// TwinCAT 3 PLC project ManRiding
// ProgramVersion: 3.1.4023.0
// libraries:
//   Tc2_ControllerToolbox, * (Beckhoff Automation GmbH)
//   Tc2_Math, * (Beckhoff Automation GmbH)
//   Tc2_MC2, * (Beckhoff Automation GmbH)
//   Tc2_MC2_Drive, * (Beckhoff Automation GmbH)
//   Tc2_ModbusSrv, * (Beckhoff Automation GmbH)
//   Tc2_SerialCom, * (Beckhoff Automation GmbH)
//   Tc2_Standard, * (Beckhoff Automation GmbH)
//   Tc2_System, * (Beckhoff Automation GmbH)
//   Tc2_TcpIp, * (Beckhoff Automation GmbH)
//   Tc2_Utilities, * (Beckhoff Automation GmbH)
//   Tc3_Database, * (Beckhoff Automation GmbH)
//   Tc3_JsonXml, * (Beckhoff Automation GmbH)
//   Tc3_Module, * (Beckhoff Automation GmbH)
//   VisuDialogs, * (System)
//   VisuSymbols, * (System)
//   VisuSymbols,3.5.10.0,System
// project tree:
//   / GlobalTextList.TcGTLO, PlcTask.TcTTO, Visualization Manager.TcVMO (not stored)
//   GVLs/ GVL.TcGVL, INPUT.TcGVL, OUTPUT.TcGVL
//   POUs/ FB_AxisControl.TcPOU, FUN_In_Zone.TcPOU, MAIN.TcPOU
//   VISUs/ Visualization.TcVIS
// real-time tasks:
//   TASK PlcTask: cycle T#10ms, priority 20, ADS port 350
// motion (NC):
//   TASK NC-Task 1 SAF: cycle T#2ms, priority 4, ADS port 501
//   TASK NC-Task 1 SVB: cycle T#10ms, priority 8, ADS port 511
//   AXIS Axis 1 (BogieDrv1) (id 1)
//     OtherSettings: AllowMotionCmdToSlave=true
//     encoder EncType=1
//     drive DrvType=5
//       Analog: TorqueSetpointScale=10, ScaleFactorActTorque=0.1
//     controller CtrType=1
//       CtrPara: PriorControlFactor=1
//         Observer: BandWidth=20
//   AXIS Axis 2 (BogieDrv2) (id 2)
//     OtherSettings: AllowMotionCmdToSlave=true
//     encoder EncType=1
//     drive DrvType=5
//       Analog: TorqueSetpointScale=10, ScaleFactorActTorque=0.1
//     controller CtrType=1
//       CtrPara: PriorControlFactor=1
//         Observer: BandWidth=20
//   AXIS Axis 3 (BogieDrv3) (id 3)
//     OtherSettings: AllowMotionCmdToSlave=true
//     encoder EncType=1
//     drive DrvType=5
//       Analog: TorqueSetpointScale=10, ScaleFactorActTorque=0.1
//     controller CtrType=1
//       CtrPara: PriorControlFactor=1
//         Observer: BandWidth=20
//   AXIS Axis 4 (BogieDrv4) (id 4)
//     OtherSettings: AllowMotionCmdToSlave=true
//     encoder EncType=1
//     drive DrvType=5
//       Analog: TorqueSetpointScale=10, ScaleFactorActTorque=0.1
//     controller CtrType=1
//       CtrPara: PriorControlFactor=1
//         Observer: BandWidth=20
//   AXIS Axis 5 (Stabiliser A) (id 5)
//     Dynamic: AccelerationMaximum=50000, DecelerationMaximum=50000, Acceleration=1371.32, Deceleration=1371.32, Jerk=1385020, FastAxisStopSignalType=4
//     Velo: RefSearch=1.357738094695, RefSync=1.357738094695, SlowManual=6.788690473475, FastManual=40.73214284085, Fast=135.7738094695, Maximum=135.774
//     OtherSettings: AllowMotionCmdToSlave=true
//     encoder EncType=19
//       EncPara: ScaleFactorNumerator=3.57142857, ScaleFactorDenominator=1048576, Offset=104.9, MaxCount=#xffffffff
//         SoftEndMinControl: Enable=true, Range=-10
//         SoftEndMaxControl: Enable=true, Range=200
//     drive DrvType=16
//       DrvPara: MaxCount=#xffffffff, DriveControlDWord=#x00020000
//         Analog: VeloReferenz=149.35119041645, VeloScale=32, TorqueSetpointScale=10, ScaleFactorActTorque=0.1
//         TimeComp: TaskDelayCycles=1
//     controller CtrType=1
//       CtrPara: PriorControlFactor=1
//         PosDiffControl: Enable=false
//         PID: PosKp=30
//         Observer: BandWidth=20
//   AXIS Axis 6 (Stabiliser B) (id 6)
//     Dynamic: AccelerationMaximum=50000, DecelerationMaximum=50000, Acceleration=1371.32, Deceleration=1371.32, Jerk=1385030, FastAxisStopSignalType=4
//     Velo: RefSearch=1.357738094695, RefSync=1.357738094695, SlowManual=6.788690473475, FastManual=40.73214284085, Fast=135.7738094695, Maximum=135.774
//     OtherSettings: AllowMotionCmdToSlave=true
//     encoder EncType=19
//       EncPara: ScaleFactorNumerator=3.57142857, ScaleFactorDenominator=1048576, Offset=411, Inverse=true, MaxCount=#xffffffff
//         SoftEndMinControl: Enable=true, Range=-10
//         SoftEndMaxControl: Enable=true, Range=200
//     drive DrvType=16
//       DrvPara: Inverse=true, MaxCount=#xffffffff, DriveControlDWord=#x00020000
//         Analog: VeloReferenz=149.35119041645, VeloScale=32, TorqueSetpointScale=10, ScaleFactorActTorque=0.1
//         TimeComp: TaskDelayCycles=1
//     controller CtrType=1
//       CtrPara: PriorControlFactor=1
//         PosDiffControl: Enable=false
//         PID: PosKp=30
//         Observer: BandWidth=20
//   AXIS Axis 7 (Stabiliser C) (id 7)
//     Dynamic: AccelerationMaximum=50000, DecelerationMaximum=50000, Acceleration=1371.32, Deceleration=1371.32, Jerk=1385030, FastAxisStopSignalType=4
//     Velo: RefSearch=1.357738094695, RefSync=1.357738094695, SlowManual=6.788690473475, FastManual=40.73214284085, Fast=135.7738094695, Maximum=135.774
//     OtherSettings: AllowMotionCmdToSlave=true
//     encoder EncType=19
//       EncPara: ScaleFactorNumerator=3.57142857, ScaleFactorDenominator=1048576, Offset=-4435, MaxCount=#xffffffff
//         SoftEndMinControl: Enable=true, Range=-10
//         SoftEndMaxControl: Enable=true, Range=200
//     drive DrvType=16
//       DrvPara: MaxCount=#xffffffff, DriveControlDWord=#x00020000
//         Analog: VeloReferenz=149.35119041645, VeloScale=32, TorqueSetpointScale=10, ScaleFactorActTorque=0.1
//         TimeComp: TaskDelayCycles=1
//     controller CtrType=1
//       CtrPara: PriorControlFactor=1
//         PosDiffControl: Enable=false
//         PID: PosKp=30
//         Observer: BandWidth=20
//   AXIS Axis 8 (Stabiliser D) (id 8)
//     Dynamic: AccelerationMaximum=50000, DecelerationMaximum=50000, Acceleration=1371.32, Deceleration=1371.32, Jerk=1385030, FastAxisStopSignalType=4
//     Velo: RefSearch=1.357738094695, RefSync=1.357738094695, SlowManual=6.788690473475, FastManual=40.73214284085, Fast=135.7738094695, Maximum=135.774
//     OtherSettings: AllowMotionCmdToSlave=true
//     encoder EncType=19
//       EncPara: ScaleFactorNumerator=3.57142857, ScaleFactorDenominator=1048576, Offset=288.9, Inverse=true, MaxCount=#xffffffff
//         SoftEndMinControl: Enable=true, Range=-10
//         SoftEndMaxControl: Enable=true, Range=200
//     drive DrvType=16
//       DrvPara: Inverse=true, MaxCount=#xffffffff
//         Analog: VeloReferenz=149.35119041645, VeloScale=32, TorqueSetpointScale=10, ScaleFactorActTorque=0.1
//         TimeComp: TaskDelayCycles=1
//     controller CtrType=1
//       CtrPara: PriorControlFactor=1
//         PosDiffControl: Enable=false
//         PID: PosKp=30
//         Observer: BandWidth=20

CONFIGURATION ManRiding
    RESOURCE PLC ON TwinCAT3
        TASK PlcTask(INTERVAL := T#10ms, PRIORITY := 20);
        PROGRAM MAIN WITH PlcTask : MAIN;
    END_RESOURCE
END_CONFIGURATION

// ---- GVLs/GVL.TcGVL
	{attribute 'qualified_only'}
	{attribute 'TcContextName':='PlcTaskMAIN'}
VAR_GLOBAL PERSISTENT
	//New Version
	Bogie_Clean_Position : REAL := 0;
		
END_VAR

VAR_GLOBAL CONSTANT
	
END_VAR


VAR_GLOBAL
	Home_Button_Activated 		: BOOL := FALSE;
	Cleaning_Button_Activated 	: BOOL := FALSE;
	Finish_Current_Brick 		: BOOL := FALSE;
	HMI_Connected 				: BOOL := FALSE;
	database		: ARRAY[0..100] OF STRING(100);(* Target PLC database *)

	
	AMSID : T_AmsNetId  := '5.61.32.144.1.1';       // this is the ADS address for the IPC on the robot

	Use_Current_As_Clean_Position : BOOL := FALSE;
	
{region "axis refs"}	
	Bogie_DriveA	: AXIS_REF; 
	Bogie_DriveB	: AXIS_REF; 
	Bogie_DriveC	: AXIS_REF; 
	Bogie_DriveD	: AXIS_REF; 		 
	Stabiliser_A_Axis	: AXIS_REF;
	Stabiliser_B_Axis	: AXIS_REF;	
	Stabiliser_C_Axis	: AXIS_REF;		
	Stabiliser_D_Axis	: AXIS_REF;		
		 
	Bogie_DriveA_Velocity        	: LREAL;
	Bogie_DriveB_Velocity        	: LREAL;
	Bogie_DriveC_Velocity        	: LREAL;
	Bogie_DriveD_Velocity        	: LREAL;

{endregion}
	 
{region "TCP/Lazer Adjust"}

{endregion}

{region "Bogie Alarm"}
	BogieAlarmTimer : TON := (PT := T#2S);
{endregion}
	
{region "procedure variables"}	
	// Main procedure Variables
	IsEnabled		   : BOOL	:= FALSE;
	Is_Running          : BOOL;                         // the boolean to indicate if the robot is running in a sequence mode
	Is_Start_Button_Pressed          : BOOL;                         // boolean representing the start button on the HMI
	Is_Stop_Button_Pressed           : BOOL := TRUE;                 // boolean representing the stop button on the HMI - boots to false, preventing the sequence initiaiting without explicit commmand
	Cancel_Manuals					 : BOOL;		 
	
{region "ablr/ bogie vars"}	
	// Four Wheel Drive Bogie System
	Bogie_Pause					: BOOL := FALSE;
	  
	Bogie_DriveA_Current_Position      : REAL;                          // bogie current position  
	Bogie_DriveA_Required_Position     : REAL;
	Bogie_DriveA_In_Position           : BOOL;
	Bogie_DriveA_Manual_Enable         : BOOL;
	Bogie_DriveA_Encoder_Reset         : BOOL := FALSE;
	Bogie_DriveA_Pause					: BOOL := FALSE;
		 
	Bogie_DriveB_Current_Position      : REAL;                          // bogie current position
	Bogie_DriveB_Required_Position     : REAL;
	Bogie_DriveB_In_Position           : BOOL;
	Bogie_DriveB_Manual_Enable         : BOOL;
	Bogie_DriveB_Encoder_Reset         : BOOL := FALSE;
	Bogie_DriveB_Pause					: BOOL := FALSE;
		 
	Bogie_DriveC_Current_Position      : REAL;                          // bogie current position
	Bogie_DriveC_Required_Position     : REAL;
	Bogie_DriveC_In_Position           : BOOL;
	Bogie_DriveC_Manual_Enable         : BOOL;
	Bogie_DriveC_Encoder_Reset         : BOOL := FALSE;
	Bogie_DriveC_Pause					: BOOL := FALSE;
		 
	Bogie_DriveD_Current_Position      : REAL;                          // bogie current position
	Bogie_DriveD_Required_Position     : REAL;
	Bogie_DriveD_In_Position           : BOOL;
	Bogie_DriveD_Manual_Enable         : BOOL;
	Bogie_DriveD_Encoder_Reset         : BOOL := FALSE;
	Bogie_DriveD_Pause					: BOOL := FALSE;

{endregion}
	
	Bogie_Stabiliser_A_Deployed :BOOL := TRUE;
	Bogie_Stabiliser_A_Deploy :BOOL := FALSE;
	Bogie_Stabiliser_A_Manual_Enable  :BOOL :=FALSE;
	Bogie_Stabiliser_A_Current_Position :REAL :=0;
	Bogie_Stabiliser_A_Required_Position :LREAL :=0;
	Bogie_Stabiliser_A_In_Position : BOOL := FALSE;

	Bogie_Stabiliser_B_Deployed :BOOL := TRUE;
	Bogie_Stabiliser_B_Deploy :BOOL := FALSE;
	Bogie_Stabiliser_B_Manual_Enable  :BOOL :=FALSE;
	Bogie_Stabiliser_B_Current_Position :REAL :=0;
	Bogie_Stabiliser_B_Required_Position :LREAL :=0;
	Bogie_Stabiliser_B_In_Position : BOOL := FALSE;

	Bogie_Stabiliser_C_Deployed :BOOL := TRUE;
	Bogie_Stabiliser_C_Deploy :BOOL := FALSE;
	Bogie_Stabiliser_C_Manual_Enable  :BOOL :=FALSE;
	Bogie_Stabiliser_C_Current_Position :REAL :=0;
	Bogie_Stabiliser_C_Required_Position :LREAL :=0;
	Bogie_Stabiliser_C_In_Position : BOOL := FALSE;

	Bogie_Stabiliser_D_Deployed :BOOL := TRUE;
	Bogie_Stabiliser_D_Deploy :BOOL := FALSE;
	Bogie_Stabiliser_D_Manual_Enable  :BOOL :=FALSE;
	Bogie_Stabiliser_D_Current_Position :REAL :=0;
	Bogie_Stabiliser_D_Required_Position :LREAL :=0;
	Bogie_Stabiliser_D_In_Position : BOOL := FALSE;
			
	Stabiliser_Max_Torque_1 :REAL := 1150;
	Stabiliser_Max_Torque_2 :REAL := -1150;
		
	Bogie_Stabiliser_B: INT;
	
	ABLR_Height	:REAL	:=0;
	ABLR_Brick_Len :REAL :=0;
	
	RawYawValue : REAL := 0;
	
	RxBufferEL			: ComBuffer;	(* Receive data buffer; used with all receive function blocks *)
	TxBufferEL			: ComBuffer;	(* Transmit data buffer; used with all receive function blocks *)
	
	Brick_Measured :BOOL := FALSE;
	
END_VAR

// ---- GVLs/INPUT.TcGVL
{attribute 'qualified_only'}
{attribute 'TcContextName':='PlcTaskMAIN'}
VAR_GLOBAL

	Is_Emergency_Stop_Healthy AT%I* : BOOL := TRUE;                    // Emergency stop boolean	

	Temperature_Sensor_Raw     AT%I* : INT := 100;									  // Temperature pulled from the LowerBoard > Term7 > RTD > Value 
	Wind_Speed_In              AT%I* : INT;                                   
	
	ABLR_Current_Position   AT%I* : UDINT;
	
	ABLR_Arm_Inclinometer_X_In AT%I* : INT;
	ABLR_Arm_Inclinometer_X : REAL;
	ABLR_Arm_Inclinometer_Y_In AT%I* : INT;
	ABLR_Arm_Inclinometer_Y : REAL;
		
	Stabilser_A_Torque			AT%I* : INT;
	Stabilser_B_Torque			AT%I* : INT;
	Stabilser_C_Torque			AT%I* : INT;
	Stabilser_D_Torque			AT%I* : INT;
	
	DriveA_Velocity				AT%I* : REAL;
	DriveB_Velocity				AT%I* : REAL;
	DriveC_Velocity				AT%I* : REAL;
	DriveD_Velocity				AT%I* : REAL;
	
	DriveA_Torque				AT%I* : INT;
	DriveB_Torque				AT%I* : INT;
	DriveC_Torque				AT%I* : INT;
	DriveD_Torque				AT%I* : INT;
		
END_VAR

// ---- GVLs/OUTPUT.TcGVL
{attribute 'qualified_only'}
{attribute 'TcContextName':='PlcTaskMAIN'}
VAR_GLOBAL

	BogieAlarmEngaged AT%Q* : BOOL;

	Bogie_Stabiliser_Hi_Speed     AT%Q* : BOOL;
	Bogie_Stabiliser_Fwd          AT%Q* : BOOL;
	Bogie_Stabiliser_Rev          AT%Q* : BOOL;
	
	Stabiliser_A_FastStop	AT%Q*	:USINT	:= 0;
	Stabiliser_B_FastStop	AT%Q*	:USINT	:= 0;
	Stabiliser_C_FastStop	AT%Q*	:USINT	:= 0;
	Stabiliser_D_FastStop	AT%Q*	:USINT	:= 0;

END_VAR

// ---- POUs/MAIN.TcPOU
PROGRAM MAIN
VAR CONSTANT
	Bogie_Allowable_Error : REAL := 2;	// Should be 0.5 - 1
	Bogie_Stabiliser_Allowable_Error : REAL := 0.5;
END_VAR
VAR	
	AmsId    : T_AmsNetId := '5.61.32.144.1.1';
	bChangeSeparatorToComma	: BOOL := FALSE;
{region "sequence timer"=======================================================
	fbSequenceTimer        : FB_Sequence_Timer;
	SequenceTimerArray     : ARRAY [0..255] OF REAL;
	ResetSequenceTimeCount : BOOL;
{endregion}
	
    fbStabiliser_Control_A     : FB_AxisControl := (fVelocity := 50);	
	fbStabiliser_Control_B     : FB_AxisControl := (fVelocity := 50);	
	fbStabiliser_Control_C     : FB_AxisControl := (fVelocity := 50);	
	fbStabiliser_Control_D    : FB_AxisControl := (fVelocity := 50);
		 
	// Four Wheel Drive Bogie System

	Bogie_DriveA_Control         	: FB_AxisControl;   // FRONT RIGHT
	Bogie_DriveA_Position	: REAL;
	 
	Bogie_DriveB_Control         	: FB_AxisControl;	//REAR RIGHT
	Bogie_DriveB_Position	: REAL;
	
	Bogie_DriveC_Control         	: FB_AxisControl;   // FRONT RIGHT
	Bogie_DriveC_Position	: REAL;
	 
	Bogie_DriveD_Control         	: FB_AxisControl;	//REAR RIGHT
	Bogie_DriveD_Position	: REAL;
		  	
	Boogie_Reset_Counter : INT := 0;
	BoogieHome : BOOL := FALSE;
	Boogie_Reset_Position : REAL := 5400;
	Bogie_Slow_Zone : REAL := 100;
	Boogie_Threshold_Crossed : BOOL := FALSE; 
	
	Bogie_Stabiliser_Slow_Zone : REAL := 10;
	
	StabAResetSent : BOOL := FALSE;
	StabBResetSent : BOOL := FALSE;
	StabCResetSent : BOOL := FALSE;
	StabDResetSent : BOOL := FALSE;
	StabiliserAResst : TON :=(PT := T#10MS);
	StabiliserBResst : TON :=(PT := T#10MS);
	StabiliserCResst : TON :=(PT := T#10MS);
	StabiliserDResst : TON :=(PT := T#10MS);
	
	BCount : INT := 0;
	Trigger_Found : BOOL := FALSE;
	
	fPosition: REAL;

END_VAR

//################################## AC axes control ############################################################################


IF (NOT GVL.Bogie_Stabiliser_A_Deployed) AND (NOT GVL.Bogie_Stabiliser_B_Deployed) AND (NOT GVL.Bogie_Stabiliser_C_Deployed) AND (NOT GVL.Bogie_Stabiliser_D_Deployed) THEN
	IF NOT (GVL.Bogie_Pause) THEN				
		
	Bogie_DriveA_Control(
		xEnable     := (GVL.IsEnabled) OR (GVL.Bogie_DriveA_Manual_Enable),
		xMoveA      := NOT GVL.Bogie_DriveA_In_Position,
		fPosition   := GVL.Bogie_DriveA_Required_Position,
		fVelocity   := GVL.Bogie_DriveA_Velocity ,
		Axis        := GVL.Bogie_DriveA);		 
			 
	GVL.Bogie_DriveA_IN_Position := FUN_In_Zone(GVL.Bogie_DriveA_Current_Position, GVL.Bogie_DriveA_Required_Position, 1);
		 
	IF(GVL.Bogie_DriveA_Manual_Enable AND GVL.Bogie_DriveA_IN_Position)THEN
	//	GVL.DriveAll := FALSE;
		GVL.Bogie_DriveA_Manual_Enable := FALSE; 
	//	GVL.Bogie_DriveB_Manual_Enable := FALSE; 
	//	GVL.Bogie_DriveC_Manual_Enable := FALSE; 
	//	GVL.Bogie_DriveD_Manual_Enable := FALSE; 
	END_IF	


	Bogie_DriveB_Control(
		xEnable     := (GVL.IsEnabled) OR (GVL.Bogie_DriveB_Manual_Enable),
		xMoveA      := NOT GVL.Bogie_DriveB_In_Position,
		fPosition   := GVL.Bogie_DriveB_Required_Position,
		fVelocity   := GVL.Bogie_DriveB_Velocity ,
		Axis        := GVL.Bogie_DriveB);		 
		 
	GVL.Bogie_DriveB_IN_Position := FUN_In_Zone(GVL.Bogie_DriveB_Current_Position, GVL.Bogie_DriveB_Required_Position, 1);
		 
	IF(GVL.Bogie_DriveB_Manual_Enable AND GVL.Bogie_DriveB_IN_Position)THEN
	//	GVL.DriveAll := FALSE;
	//	GVL.Bogie_DriveA_Manual_Enable := FALSE; 
		GVL.Bogie_DriveB_Manual_Enable := FALSE; 
	//	GVL.Bogie_DriveC_Manual_Enable := FALSE; 
	//	GVL.Bogie_DriveD_Manual_Enable := FALSE; 
	END_IF
	
	Bogie_DriveC_Control(
		xEnable     := (GVL.IsEnabled) OR (GVL.Bogie_DriveC_Manual_Enable),
		xMoveA      := NOT GVL.Bogie_DriveC_In_Position,
		fPosition   := GVL.Bogie_DriveC_Required_Position,
		fVelocity   := GVL.Bogie_DriveC_Velocity ,
		Axis        := GVL.Bogie_DriveC);		 
			 
	GVL.Bogie_DriveC_IN_Position := FUN_In_Zone(GVL.Bogie_DriveC_Current_Position, GVL.Bogie_DriveC_Required_Position, 1);
	 
	IF(GVL.Bogie_DriveB_Manual_Enable AND GVL.Bogie_DriveB_IN_Position)THEN
	//	GVL.DriveAll := FALSE;
	//	GVL.Bogie_DriveA_Manual_Enable := FALSE; 
	//	GVL.Bogie_DriveB_Manual_Enable := FALSE; 
		GVL.Bogie_DriveC_Manual_Enable := FALSE; 
	//	GVL.Bogie_DriveD_Manual_Enable := FALSE; 
	END_IF

	Bogie_DriveD_Control(
		xEnable     := (GVL.IsEnabled) OR (GVL.Bogie_DriveD_Manual_Enable),
		xMoveA      := NOT GVL.Bogie_DriveD_In_Position,
		fPosition   := GVL.Bogie_DriveD_Required_Position,
		fVelocity   := GVL.Bogie_DriveD_Velocity ,
		Axis        := GVL.Bogie_DriveD);		 
			 
	GVL.Bogie_DriveD_IN_Position := FUN_In_Zone(GVL.Bogie_DriveD_Current_Position, GVL.Bogie_DriveD_Required_Position, 1);
	 
	IF(GVL.Bogie_DriveB_Manual_Enable AND GVL.Bogie_DriveB_IN_Position)THEN
	//	GVL.DriveAll := FALSE;
	//	GVL.Bogie_DriveA_Manual_Enable := FALSE; 
	//	GVL.Bogie_DriveB_Manual_Enable := FALSE; 
	//	GVL.Bogie_DriveC_Manual_Enable := FALSE; 
		GVL.Bogie_DriveD_Manual_Enable := FALSE; 
	END_IF
	
	END_IF

ELSE
	GVL.Bogie_Stabiliser_A_Required_Position := 0;	
	GVL.Bogie_Stabiliser_A_Deploy := TRUE;
	GVL.Bogie_Stabiliser_B_Required_Position := 0;	
	GVL.Bogie_Stabiliser_B_Deploy := TRUE;	
	GVL.Bogie_Stabiliser_C_Required_Position := 0;	
	GVL.Bogie_Stabiliser_C_Deploy := TRUE;	
	//GVL.Bogie_Stabiliser_D_Required_Position := 0;	
	//GVL.Bogie_Stabiliser_D_Deploy := TRUE;	
END_IF

//-------------------------------------------------------------------------------------------------------------------

IF (GVL.Bogie_Stabiliser_A_Deploy OR GVL.Bogie_Stabiliser_A_Manual_Enable) THEN
	IF (GVL.Bogie_Stabiliser_A_Deployed) THEN
		GVL.Bogie_Stabiliser_A_Required_Position := 0;	
		GVL.Bogie_Stabiliser_A_Deployed := FALSE;	
	END_IF

	fbStabiliser_Control_A(
		xEnable := GVL.Bogie_Stabiliser_A_Manual_Enable OR GVL.Bogie_Stabiliser_A_Deploy,
		fPosition := GVL.Bogie_Stabiliser_A_Required_Position,
		xMoveA := NOT GVL.Bogie_Stabiliser_A_In_Position,
		Axis := GVL.Stabiliser_A_Axis);

	GVL.Bogie_Stabiliser_A_In_Position := FUN_In_Zone(Current := GVL.Bogie_Stabiliser_A_Current_Position, Required := GVL.Bogie_Stabiliser_A_Required_Position, Margin := 1 );	

	IF (INPUT.Stabilser_A_Torque > GVL.Stabiliser_Max_Torque_1 AND GVL.Bogie_Stabiliser_A_Required_Position > 0) THEN
		GVL.Bogie_Stabiliser_A_In_Position := TRUE;
		OUTPUT.Stabiliser_A_FastStop := 128;
		GVL.Bogie_Stabiliser_A_Required_Position := GVL.Bogie_Stabiliser_A_Current_Position;
		GVL.Bogie_Stabiliser_A_Deployed := TRUE;
		GVL.Bogie_Stabiliser_A_Deploy := FALSE;	
		GVL.Bogie_Stabiliser_A_Manual_Enable := FALSE;	
		GVL.Bogie_Stabiliser_A_Required_Position := 0;
		fbStabiliser_Control_A(
			xEnable := FALSE,
			xMoveA := FALSE,
			Axis := GVL.Stabiliser_A_Axis);	
	ELSIF (GVL.Bogie_Stabiliser_A_In_Position) THEN	
		OUTPUT.Stabiliser_A_FastStop := 128;
		IF (GVL.Bogie_Stabiliser_A_Current_Position > 100) THEN
			GVL.Bogie_Stabiliser_A_Deployed := TRUE;
		ELSE
			GVL.Bogie_Stabiliser_A_Deployed := FALSE;
		END_IF				
		GVL.Bogie_Stabiliser_A_Deploy := FALSE;		
		GVL.Bogie_Stabiliser_A_Manual_Enable := FALSE;
		GVL.Bogie_Stabiliser_A_Required_Position := 0;
		fbStabiliser_Control_A(
			xEnable := FALSE,
			xMoveA := FALSE,
			Axis := GVL.Stabiliser_A_Axis);	
	ELSIF (GVL.Bogie_Stabiliser_A_Current_Position < 60) THEN
		GVL.Bogie_Stabiliser_A_Deployed := FALSE;
	END_IF	
END_IF

IF (GVL.Bogie_Stabiliser_B_Deploy OR GVL.Bogie_Stabiliser_B_Manual_Enable) THEN
	IF (GVL.Bogie_Stabiliser_B_Deployed) THEN
		GVL.Bogie_Stabiliser_B_Required_Position := 0;	
		GVL.Bogie_Stabiliser_B_Deployed := FALSE;
	END_IF

	fbStabiliser_Control_B(
		xEnable := GVL.Bogie_Stabiliser_B_Manual_Enable OR GVL.Bogie_Stabiliser_B_Deploy,
		fPosition := GVL.Bogie_Stabiliser_B_Required_Position,
		xMoveA := NOT GVL.Bogie_Stabiliser_B_In_Position,
		Axis := GVL.Stabiliser_B_Axis);
		
	GVL.Bogie_Stabiliser_B_In_Position := FUN_In_Zone(Current := GVL.Bogie_Stabiliser_B_Current_Position, Required := GVL.Bogie_Stabiliser_B_Required_Position, Margin := 1 );	
	
	IF (INPUT.Stabilser_B_Torque < GVL.Stabiliser_Max_Torque_2 AND GVL.Bogie_Stabiliser_B_Required_Position > 0) THEN
		GVL.Bogie_Stabiliser_B_In_Position := TRUE;
		OUTPUT.Stabiliser_B_FastStop := 128;
		GVL.Bogie_Stabiliser_B_Required_Position := GVL.Bogie_Stabiliser_B_Current_Position;
		GVL.Bogie_Stabiliser_B_Deployed := TRUE;
		GVL.Bogie_Stabiliser_B_Deploy := FALSE;
		GVL.Bogie_Stabiliser_B_Manual_Enable := FALSE;
		GVL.Bogie_Stabiliser_B_Required_Position := 0;	
		fbStabiliser_Control_B(
			xEnable := FALSE,
			xMoveA := FALSE,
			Axis := GVL.Stabiliser_B_Axis);		
	ELSIF (GVL.Bogie_Stabiliser_B_In_Position) THEN	
		OUTPUT.Stabiliser_B_FastStop := 128;	
		IF (GVL.Bogie_Stabiliser_B_Current_Position > 100) THEN
			GVL.Bogie_Stabiliser_B_Deployed := TRUE;
		ELSE
			GVL.Bogie_Stabiliser_B_Deployed := FALSE;
		END_IF	
		GVL.Bogie_Stabiliser_B_Deploy := FALSE;
		GVL.Bogie_Stabiliser_B_Manual_Enable := FALSE;
		GVL.Bogie_Stabiliser_B_Required_Position := 0;	
		fbStabiliser_Control_B(
			xEnable := FALSE,
			xMoveA := FALSE,
			Axis := GVL.Stabiliser_B_Axis);			
		ELSIF (GVL.Bogie_Stabiliser_B_Current_Position < 60) THEN
		GVL.Bogie_Stabiliser_B_Deployed := FALSE;
	END_IF	
	
END_IF

IF (GVL.Bogie_Stabiliser_C_Deploy OR GVL.Bogie_Stabiliser_C_Manual_Enable) THEN
	IF (GVL.Bogie_Stabiliser_C_Deployed) THEN
		GVL.Bogie_Stabiliser_C_Required_Position := 0;	
		GVL.Bogie_Stabiliser_C_Deployed := FALSE;	
	END_IF

	fbStabiliser_Control_C(
		xEnable := GVL.Bogie_Stabiliser_C_Manual_Enable OR GVL.Bogie_Stabiliser_C_Deploy,
		fPosition := GVL.Bogie_Stabiliser_C_Required_Position,
		xMoveA := NOT GVL.Bogie_Stabiliser_C_In_Position,
		Axis := GVL.Stabiliser_C_Axis);

	GVL.Bogie_Stabiliser_C_In_Position := FUN_In_Zone(Current := GVL.Bogie_Stabiliser_C_Current_Position, Required := GVL.Bogie_Stabiliser_C_Required_Position, Margin := 1 );	

	IF (INPUT.Stabilser_C_Torque > GVL.Stabiliser_Max_Torque_1 AND GVL.Bogie_Stabiliser_C_Required_Position > 0) THEN
		GVL.Bogie_Stabiliser_C_In_Position := TRUE;
		OUTPUT.Stabiliser_C_FastStop := 128;
		GVL.Bogie_Stabiliser_C_Required_Position := GVL.Bogie_Stabiliser_C_Current_Position;
		GVL.Bogie_Stabiliser_C_Deployed := TRUE;
		GVL.Bogie_Stabiliser_C_Deploy := FALSE;	
		GVL.Bogie_Stabiliser_C_Manual_Enable := FALSE;
		GVL.Bogie_Stabiliser_C_Required_Position := 0;
		fbStabiliser_Control_C(
			xEnable := FALSE,
			xMoveA := FALSE,
			Axis := GVL.Stabiliser_C_Axis);	
	ELSIF (GVL.Bogie_Stabiliser_C_In_Position) THEN	
		OUTPUT.Stabiliser_C_FastStop := 128;				
		IF (GVL.Bogie_Stabiliser_C_Current_Position > 100) THEN
			GVL.Bogie_Stabiliser_C_Deployed := TRUE;
		ELSE
			GVL.Bogie_Stabiliser_C_Deployed := FALSE;
		END_IF	
		GVL.Bogie_Stabiliser_C_Deploy := FALSE;		
		GVL.Bogie_Stabiliser_C_Manual_Enable := FALSE;
		GVL.Bogie_Stabiliser_C_Required_Position := 0;
		fbStabiliser_Control_C(
			xEnable := FALSE,
			xMoveA := FALSE,
			Axis := GVL.Stabiliser_C_Axis);
		ELSIF (GVL.Bogie_Stabiliser_C_Current_Position < 60) THEN
		GVL.Bogie_Stabiliser_C_Deployed := FALSE;
	END_IF		
END_IF


IF (GVL.Bogie_Stabiliser_D_Deploy OR GVL.Bogie_Stabiliser_D_Manual_Enable) THEN
	IF (GVL.Bogie_Stabiliser_D_Deployed) THEN	
		GVL.Bogie_Stabiliser_D_Required_Position := 0;	
		GVL.Bogie_Stabiliser_D_Deployed := FALSE;
	END_IF
	
	fbStabiliser_Control_D(
		xEnable := GVL.Bogie_Stabiliser_D_Manual_Enable OR GVL.Bogie_Stabiliser_D_Deploy,
		fPosition := GVL.Bogie_Stabiliser_D_Required_Position,
		xMoveA := NOT GVL.Bogie_Stabiliser_D_In_Position,
		Axis := GVL.Stabiliser_D_Axis);
		
	GVL.Bogie_Stabiliser_D_In_Position := FUN_In_Zone(Current := GVL.Bogie_Stabiliser_D_Current_Position, Required := GVL.Bogie_Stabiliser_D_Required_Position, Margin := 1 );			

	IF (INPUT.Stabilser_D_Torque < GVL.Stabiliser_Max_Torque_2 AND GVL.Bogie_Stabiliser_D_Required_Position > 0) THEN
		GVL.Bogie_Stabiliser_D_In_Position := TRUE;
		OUTPUT.Stabiliser_D_FastStop := 128;
		GVL.Bogie_Stabiliser_D_Required_Position := GVL.Bogie_Stabiliser_D_Current_Position;
		GVL.Bogie_Stabiliser_D_Deployed := TRUE;
		GVL.Bogie_Stabiliser_D_Deploy := FALSE;	
		GVL.Bogie_Stabiliser_D_Manual_Enable := FALSE;
		GVL.Bogie_Stabiliser_D_Required_Position := 0;
		fbStabiliser_Control_D(
			xEnable := FALSE,
			xMoveA := FALSE,
			Axis := GVL.Stabiliser_D_Axis);	
	ELSIF (GVL.Bogie_Stabiliser_D_In_Position) THEN	
		OUTPUT.Stabiliser_D_FastStop := 128;				
		IF (GVL.Bogie_Stabiliser_D_Current_Position > 100) THEN
			GVL.Bogie_Stabiliser_D_Deployed := TRUE;
		ELSE
			GVL.Bogie_Stabiliser_D_Deployed := FALSE;
		END_IF	
		GVL.Bogie_Stabiliser_D_Deploy := FALSE;		
		GVL.Bogie_Stabiliser_D_Manual_Enable := FALSE;
		GVL.Bogie_Stabiliser_D_Required_Position := 0;
		fbStabiliser_Control_D(
			xEnable := FALSE,
			xMoveA := FALSE,
			Axis := GVL.Stabiliser_D_Axis);
		ELSIF (GVL.Bogie_Stabiliser_D_Current_Position < 60) THEN
		GVL.Bogie_Stabiliser_D_Deployed := FALSE;
	END_IF		
	
END_IF

StabiliserAResst();
StabiliserBResst();
StabiliserCResst();
StabiliserDResst();

IF ((OUTPUT.Stabiliser_A_FastStop = 128) AND  NOT StabAResetSent) THEN
	StabAResetSent := TRUE;
	StabiliserAResst.PT := T#10MS;
	StabiliserAResst.IN := TRUE;
END_IF

IF (StabiliserAResst.Q) THEN
	StabiliserAResst.IN :=FALSE;
	StabAResetSent := FALSE;
	OUTPUT.Stabiliser_A_FastStop := 0;
END_IF

IF ((OUTPUT.Stabiliser_B_FastStop = 128) AND  NOT StabBResetSent) THEN
	StabBResetSent := TRUE;
	StabiliserBResst.PT := T#10MS;
	StabiliserBResst.IN := TRUE;
END_IF

IF (StabiliserBResst.Q) THEN
	StabiliserBResst.IN :=FALSE;
	StabBResetSent := FALSE;
	OUTPUT.Stabiliser_B_FastStop := 0;
END_IF

IF ((OUTPUT.Stabiliser_C_FastStop = 128) AND  NOT StabCResetSent) THEN
	StabCResetSent := TRUE;
	StabiliserCResst.PT := T#10MS;
	StabiliserCResst.IN := TRUE;
END_IF

IF (StabiliserCResst.Q) THEN
	StabiliserCResst.IN :=FALSE;
	StabCResetSent := FALSE;
	OUTPUT.Stabiliser_C_FastStop := 0;
END_IF

IF ((OUTPUT.Stabiliser_D_FastStop = 128) AND  NOT StabDResetSent) THEN
	StabDResetSent := TRUE;
	StabiliserDResst.PT := T#10MS;
	StabiliserDResst.IN := TRUE;
END_IF

IF (StabiliserDResst.Q) THEN
	StabiliserDResst.IN :=FALSE;
	StabDResetSent := FALSE;
	OUTPUT.Stabiliser_D_FastStop := 0;
END_IF

END_PROGRAM

// ---- POUs/FB_AxisControl.TcPOU
FUNCTION_BLOCK FB_AxisControl
VAR_INPUT
	xEnable: BOOL;
	xZero: BOOL;
	xMoveR: BOOL;
	xMoveA: BOOL;
	xMoveV: BOOL;
	xPositiveDirection: BOOL;
	fDistance: LREAL;
	fPosition: LREAL;
	fVelocity: LREAL;
	xStop: BOOL;
	xHome: BOOL;
	fHomeOffset: LREAL;
	xHomeFlag: BOOL;
END_VAR
VAR_OUTPUT
	fActualPosition: LREAL;
	fActualVelocity: LREAL;
	fActModuloPos: LREAL;
	xEnabled: BOOL;
	xMoveComplete: BOOL;
	xInPosition: BOOL;
	xAtSpeed: BOOL;
	xStopped: BOOL;
	xHomed: BOOL;
	stStatus : ST_AxisStatus;
	CommandAborted : BOOL;
	bStandStill : BOOL;
END_VAR
VAR
	mcPower: MC_Power;
	mcReset: MC_Reset;
	mcMoveRelative: MC_MoveRelative;
	mcSetPosition: MC_SetPosition;
	mcMoveAbsolute: MC_MoveAbsolute;
	mcReadStatus: MC_ReadStatus;
	mcMoveVelocity: MC_MoveVelocity;
	mcStop: MC_Stop;
	mcHome: MC_Home;
END_VAR
VAR_IN_OUT
	Axis: AXIS_REF;
END_VAR

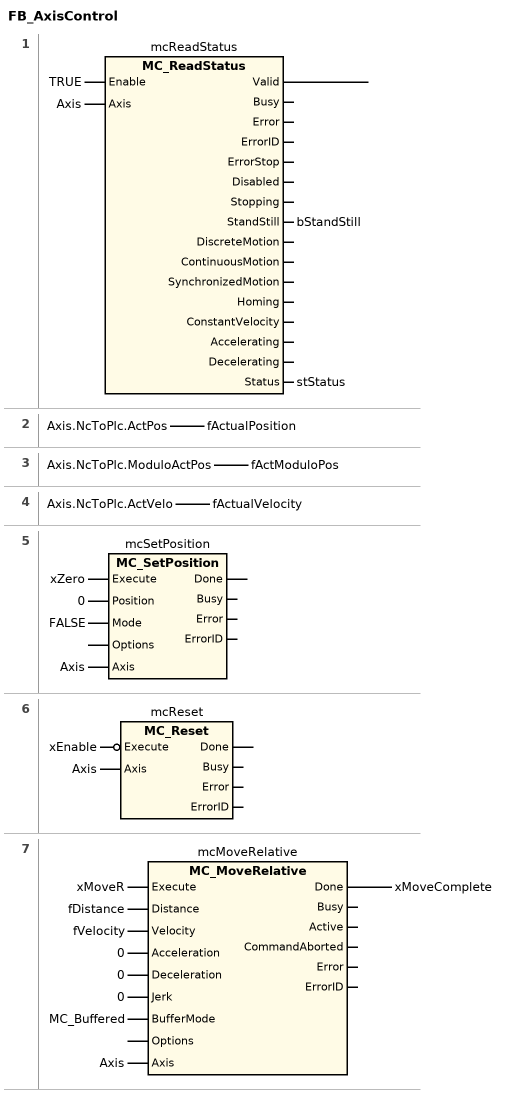
// NETWORK 1
mcReadStatus(Enable := TRUE, Axis := Axis, StandStill => bStandStill, Status => stStatus); // MC_ReadStatus

// NETWORK 2
fActualPosition := Axis.NcToPlc.ActPos;

// NETWORK 3
fActModuloPos := Axis.NcToPlc.ModuloActPos;

// NETWORK 4
fActualVelocity := Axis.NcToPlc.ActVelo;

// NETWORK 5
mcSetPosition(Execute := xZero, Position := 0, Mode := FALSE, Axis := Axis); // MC_SetPosition

// NETWORK 6
mcReset(Execute := NOT xEnable, Axis := Axis); // MC_Reset

// NETWORK 7
mcMoveRelative(
    Execute := xMoveR,
    Distance := fDistance,
    Velocity := fVelocity,
    Acceleration := 0,
    Deceleration := 0,
    Jerk := 0,
    BufferMode := MC_Buffered,
    Axis := Axis); // MC_MoveRelative
xMoveComplete := mcMoveRelative.Done;

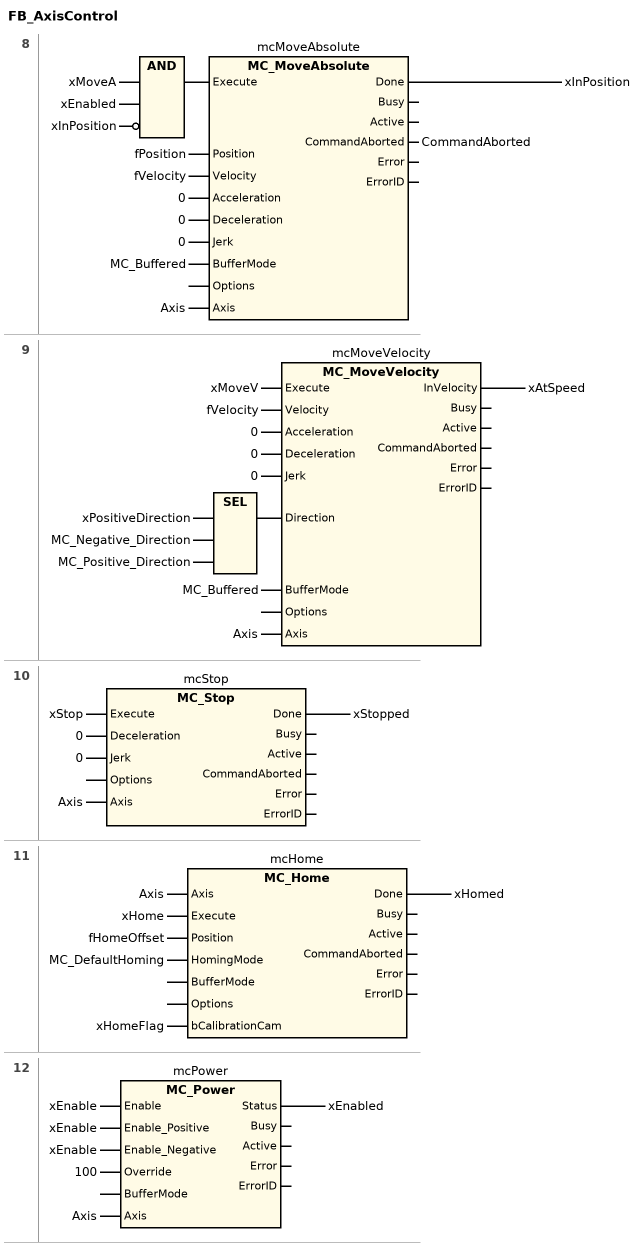
// NETWORK 8
mcMoveAbsolute(
    Execute := xMoveA AND xEnabled AND NOT xInPosition,
    Position := fPosition,
    Velocity := fVelocity,
    Acceleration := 0,
    Deceleration := 0,
    Jerk := 0,
    BufferMode := MC_Buffered,
    Axis := Axis,
    CommandAborted => CommandAborted); // MC_MoveAbsolute
xInPosition := mcMoveAbsolute.Done;

// NETWORK 9
mcMoveVelocity(
    Execute := xMoveV,
    Velocity := fVelocity,
    Acceleration := 0,
    Deceleration := 0,
    Jerk := 0,
    Direction := SEL(xPositiveDirection, MC_Negative_Direction, MC_Positive_Direction),
    BufferMode := MC_Buffered,
    Axis := Axis); // MC_MoveVelocity
xAtSpeed := mcMoveVelocity.InVelocity;

// NETWORK 10
mcStop(Execute := xStop, Deceleration := 0, Jerk := 0, Axis := Axis); // MC_Stop
xStopped := mcStop.Done;

// NETWORK 11
mcHome(
    Axis := Axis,
    Execute := xHome,
    Position := fHomeOffset,
    HomingMode := MC_DefaultHoming,
    bCalibrationCam := xHomeFlag); // MC_Home
xHomed := mcHome.Done;

// NETWORK 12
mcPower(
    Enable := xEnable,
    Enable_Positive := xEnable,
    Enable_Negative := xEnable,
    Override := 100,
    Axis := Axis); // MC_Power
xEnabled := mcPower.Status;

END_FUNCTION_BLOCK

// ---- POUs/FUN_In_Zone.TcPOU
FUNCTION FUN_In_Zone : BOOL
VAR_INPUT
	Current  : LREAL;
	Required : LREAL;
	Margin    : LREAL;
END_VAR
VAR
END_VAR

IF ((Current) < (Required + Margin )) AND ((Current) > (Required - Margin)) THEN
	FUN_In_Zone := TRUE;
ELSE
	FUN_In_Zone := FALSE;
END_IF

END_FUNCTION

// ---- GlobalTextList.TcGTLO
TEXTLIST GlobalTextList
  893 = '%f'
  263 = '+'
  904 = '+ +'
  718 = '-'
  863 = '- -'
  553 = 'Bogie Drive 1'
  807 = 'Bogie Drive 3'
  138 = 'Bogie Drive 4'
  745 = 'Bogie Drvie 2'
  1232 = 'Deploy A'
  811 = 'Deploy B'
  594 = 'Deploy C'
  767 = 'Deploy D'
  69 = 'Enable'
  22 = 'Power'
  1415 = 'Stab_A'
  1651 = 'Stab_B'
  1484 = 'Stab_C'
  1215 = 'Stab_D'
END_TEXTLIST

// ---- VISUs/Visualization.TcVIS
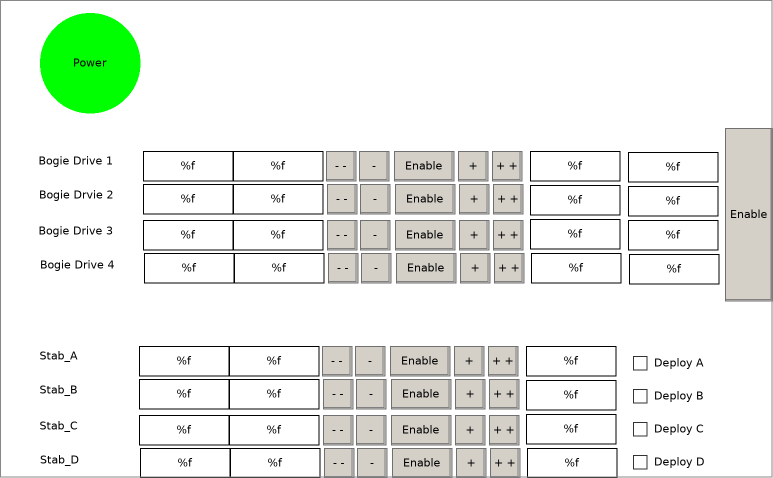
VISUALIZATION Visualization  // 773x478
    Label (25,341 67x30), "Stab_A"
    Rectangle (139,346 90x30), "%f", text variable: GVL.Bogie_Stabiliser_A_Current_Position, colour toggle: GVL.Gripper_In_Position
    Rectangle (229,346 90x30), "%f", text variable: GVL.Bogie_Stabiliser_A_Required_Position
        OnMouseUp: change screen: VisuDialogs.Numpad
    Button (355,346 30x30), "-"
        OnMouseUp: execute { GVL.Bogie_Stabiliser_A_Required_Position := GVL.Bogie_Stabiliser_A_Required_Position - 1; }
    Button (454,346 30x30), "+"
        OnMouseUp: execute { GVL.Bogie_Stabiliser_A_Required_Position := GVL.Bogie_Stabiliser_A_Required_Position + 1; }
    Button (322,346 30x30), "- -"
        OnMouseUp: execute { GVL.Bogie_Stabiliser_A_Required_Position := GVL.Bogie_Stabiliser_A_Required_Position - 10; }
    Button (488,346 30x30), "+ +"
        OnMouseUp: execute { GVL.Bogie_Stabiliser_A_Required_Position := GVL.Bogie_Stabiliser_A_Required_Position + 10; }
    Button (390,346 60x30), "Enable"
        tap GVL.Bogie_Stabiliser_A_Manual_Enable
    Label (25,375 67x30), "Stab_B"
    Rectangle (139,379 90x30), "%f", text variable: GVL.Bogie_Stabiliser_B_Current_Position, colour toggle: GVL.Gripper_In_Position
    Rectangle (229,379 90x30), "%f", text variable: GVL.Bogie_Stabiliser_B_Required_Position
        OnMouseUp: change screen: VisuDialogs.Numpad
    Button (356,379 30x30), "-"
        OnMouseUp: execute { GVL.Bogie_Stabiliser_B_Required_Position := GVL.Bogie_Stabiliser_B_Required_Position - 1; }
    Button (455,379 30x30), "+"
        OnMouseUp: execute { GVL.Bogie_Stabiliser_B_Required_Position := GVL.Bogie_Stabiliser_B_Required_Position + 1; }
    Button (323,379 30x30), "- -"
        OnMouseUp: execute { GVL.Bogie_Stabiliser_B_Required_Position := GVL.Bogie_Stabiliser_B_Required_Position - 10; }
    Button (489,379 30x30), "+ +"
        OnMouseUp: execute { GVL.Bogie_Stabiliser_B_Required_Position := GVL.Bogie_Stabiliser_B_Required_Position + 10; }
    Button (391,379 60x30), "Enable"
        tap GVL.Bogie_Stabiliser_B_Manual_Enable
    Label (25,411 67x30), "Stab_C"
    Rectangle (139,415 90x30), "%f", text variable: GVL.Bogie_Stabiliser_C_Current_Position, colour toggle: GVL.Gripper_In_Position
    Rectangle (229,415 90x30), "%f", text variable: GVL.Bogie_Stabiliser_C_Required_Position
        OnMouseUp: change screen: VisuDialogs.Numpad
    Button (356,415 30x30), "-"
        OnMouseUp: execute { GVL.Bogie_Stabiliser_C_Required_Position := GVL.Bogie_Stabiliser_C_Required_Position - 1; }
    Button (455,415 30x30), "+"
        OnMouseUp: execute { GVL.Bogie_Stabiliser_C_Required_Position := GVL.Bogie_Stabiliser_C_Required_Position + 1; }
    Button (323,415 30x30), "- -"
        OnMouseUp: execute { GVL.Bogie_Stabiliser_C_Required_Position := GVL.Bogie_Stabiliser_C_Required_Position - 10; }
    Button (489,415 30x30), "+ +"
        OnMouseUp: execute { GVL.Bogie_Stabiliser_C_Required_Position := GVL.Bogie_Stabiliser_C_Required_Position + 10; }
    Button (391,415 60x30), "Enable"
        tap GVL.Bogie_Stabiliser_C_Manual_Enable
    Label (26,445 67x30), "Stab_D"
    Rectangle (140,448 90x30), "%f", text variable: GVL.Bogie_Stabiliser_D_Current_Position, colour toggle: GVL.Gripper_In_Position
    Rectangle (230,448 90x30), "%f", text variable: GVL.Bogie_Stabiliser_D_Required_Position
        OnMouseUp: change screen: VisuDialogs.Numpad
    Button (357,448 30x30), "-"
        OnMouseUp: execute { GVL.Bogie_Stabiliser_D_Required_Position := GVL.Bogie_Stabiliser_D_Required_Position - 1; }
    Button (456,448 30x30), "+"
        OnMouseUp: execute { GVL.Bogie_Stabiliser_D_Required_Position := GVL.Bogie_Stabiliser_D_Required_Position + 1; }
    Button (324,448 30x30), "- -"
        OnMouseUp: execute { GVL.Bogie_Stabiliser_D_Required_Position := GVL.Bogie_Stabiliser_D_Required_Position - 10; }
    Button (490,448 30x30), "+ +"
        OnMouseUp: execute { GVL.Bogie_Stabiliser_D_Required_Position := GVL.Bogie_Stabiliser_D_Required_Position + 10; }
    Button (392,448 60x30), "Enable"
        tap GVL.Bogie_Stabiliser_D_Manual_Enable
    Rectangle (526,346 90x30), "%f", text variable: INPUT.Stabilser_A_Torque, colour toggle: GVL.Gripper_In_Position
    Rectangle (526,380 90x30), "%f", text variable: INPUT.Stabilser_B_Torque, colour toggle: GVL.Gripper_In_Position
    Rectangle (526,414 90x30), "%f", text variable: INPUT.Stabilser_C_Torque, colour toggle: GVL.Gripper_In_Position
    Rectangle (527,448 90x30), "%f", text variable: INPUT.Stabilser_D_Torque, colour toggle: GVL.Gripper_In_Position
    Checkbox (631,348 131x30), "Deploy A", variable: GVL.Bogie_Stabiliser_A_Deploy
    Checkbox (631,381 131x30), "Deploy B", variable: GVL.Bogie_Stabiliser_B_Deploy
    Checkbox (631,414 131x30), "Deploy C", variable: GVL.Bogie_Stabiliser_C_Deploy
    Checkbox (631,447 131x30), "Deploy D", variable: GVL.Bogie_Stabiliser_D_Deploy
    Label (29,146 94x30), "Bogie Drive 1"
    Rectangle (143,151 90x30), "%f", text variable: GVL.Bogie_DriveA_Current_Position, colour toggle: GVL.Gripper_In_Position
    Rectangle (233,151 90x30), "%f", text variable: GVL.Bogie_DriveA_Required_Position
        OnMouseUp: change screen: VisuDialogs.Numpad
    Button (359,151 30x30), "-"
        OnMouseUp: execute { GVL.Bogie_DriveA_Required_Position := GVL.Bogie_DriveA_Required_Position - 1; }
    Button (458,151 30x30), "+"
        OnMouseUp: execute { GVL.Bogie_DriveA_Required_Position := GVL.Bogie_DriveA_Required_Position + 1; }
    Button (326,151 30x30), "- -"
        OnMouseUp: execute { GVL.Bogie_DriveA_Required_Position := GVL.Bogie_DriveA_Required_Position - 10; }
    Button (492,151 30x30), "+ +"
        OnMouseUp: execute { GVL.Bogie_DriveA_Required_Position := GVL.Bogie_DriveA_Required_Position + 10; }
    Button (394,151 60x30), "Enable"
        tap GVL.Bogie_DriveA_Manual_Enable
    Label (29,180 95x30), "Bogie Drvie 2"
    Rectangle (143,184 90x30), "%f", text variable: GVL.Bogie_DriveB_Current_Position, colour toggle: GVL.Gripper_In_Position
    Rectangle (233,184 90x30), "%f", text variable: GVL.Bogie_DriveB_Required_Position
        OnMouseUp: change screen: VisuDialogs.Numpad
    Button (360,184 30x30), "-"
        OnMouseUp: execute { GVL.Bogie_DriveB_Required_Position := GVL.Bogie_DriveB_Required_Position - 1; }
    Button (459,184 30x30), "+"
        OnMouseUp: execute { GVL.Bogie_DriveB_Required_Position := GVL.Bogie_DriveB_Required_Position + 1; }
    Button (327,184 30x30), "- -"
        OnMouseUp: execute { GVL.Bogie_DriveB_Required_Position := GVL.Bogie_DriveB_Required_Position - 10; }
    Button (493,184 30x30), "+ +"
        OnMouseUp: execute { GVL.Bogie_DriveB_Required_Position := GVL.Bogie_DriveB_Required_Position + 10; }
    Button (395,184 60x30), "Enable"
        tap GVL.Bogie_DriveB_Manual_Enable p1329445385=TRUE
    Label (29,216 94x30), "Bogie Drive 3"
    Rectangle (143,220 90x30), "%f", text variable: GVL.Bogie_DriveC_Current_Position, colour toggle: GVL.Gripper_In_Position
    Rectangle (233,220 90x30), "%f", text variable: GVL.Bogie_Stabiliser_C_Required_Position
        OnMouseUp: change screen: VisuDialogs.Numpad
    Button (360,220 30x30), "-"
        OnMouseUp: execute { GVL.Bogie_Stabiliser_C_Required_Position := GVL.Bogie_Stabiliser_C_Required_Position - 1; }
    Button (459,220 30x30), "+"
        OnMouseUp: execute { GVL.Bogie_Stabiliser_C_Required_Position := GVL.Bogie_Stabiliser_C_Required_Position + 1; }
    Button (327,220 30x30), "- -"
        OnMouseUp: execute { GVL.Bogie_DriveC_Required_Position := GVL.Bogie_DriveC_Required_Position - 10; }
    Button (493,220 30x30), "+ +"
        OnMouseUp: execute { GVL.Bogie_DriveC_Required_Position := GVL.Bogie_DriveC_Required_Position + 10; }
    Button (395,220 60x30), "Enable"
        tap GVL.Bogie_DriveC_Manual_Enable
    Label (30,250 95x30), "Bogie Drive 4"
    Rectangle (144,253 90x30), "%f", text variable: GVL.Bogie_DriveD_Current_Position, colour toggle: GVL.Gripper_In_Position
    Rectangle (234,253 90x30), "%f", text variable: GVL.Bogie_Stabiliser_D_Required_Position
        OnMouseUp: change screen: VisuDialogs.Numpad
    Button (361,253 30x30), "-"
        OnMouseUp: execute { GVL.Bogie_Stabiliser_D_Required_Position := GVL.Bogie_Stabiliser_D_Required_Position - 1; }
    Button (460,253 30x30), "+"
        OnMouseUp: execute { GVL.Bogie_Stabiliser_D_Required_Position := GVL.Bogie_Stabiliser_D_Required_Position + 1; }
    Button (328,253 30x30), "- -"
        OnMouseUp: execute { GVL.Bogie_DriveD_Required_Position := GVL.Bogie_DriveD_Required_Position - 10; }
    Button (494,253 30x30), "+ +"
        OnMouseUp: execute { GVL.Bogie_Stabiliser_D_Required_Position := GVL.Bogie_Stabiliser_D_Required_Position + 10; }
    Button (396,253 60x30), "Enable"
        tap GVL.Bogie_DriveD_Manual_Enable
    Rectangle (530,151 90x30), "%f", text variable: GVL.Drive_A_Velocity, colour toggle: GVL.Gripper_In_Position
    Rectangle (530,185 90x30), "%f", text variable: GVL.Drive_B_Velocity, colour toggle: GVL.Gripper_In_Position
    Rectangle (530,219 90x30), "%f", text variable: GVL.Drive_C_Velocity, colour toggle: GVL.Gripper_In_Position
    Rectangle (531,253 90x30), "%f", text variable: GVL.Drive_D_Velocity, colour toggle: GVL.Gripper_In_Position
    Button (725,128 48x173), "Enable"
        toggle GVL.DriveAll
    Rectangle (628,152 90x30), "%f", text variable: INPUT.DriveA_Torque, colour toggle: GVL.Gripper_In_Position
    Rectangle (628,186 90x30), "%f", text variable: INPUT.DriveB_Torque, colour toggle: GVL.Gripper_In_Position
    Rectangle (628,220 90x30), "%f", text variable: INPUT.DriveC_Torque, colour toggle: GVL.Gripper_In_Position
    Rectangle (629,254 90x30), "%f", text variable: INPUT.DriveD_Torque, colour toggle: GVL.Gripper_In_Position
    Ellipse (40,13 100x100), "Power", colour toggle: (NOT INPUT.Is_Emergency_Stop_Healthy)
        toggle Input.Is_Emergency_Stop_Healthy
END_VISUALIZATION
